PROGRAM P_DecSollRuettel
VAR
END_VAR

IF DB6.iSortierer > 0 THEN
	DB6.iSortierer := DB6.iSortierer - 1;
END_IF

END_PROGRAM

(* stored: Version 1.1.0.1, ProductVersion 3.1.4024.3
   POU P_DecSollRuettel: Id {82c7bec7-7d15-4e8b-b32f-d2d38691dd47}, SpecialFunc None *)
